{attribute 'GeneratedUsingTerminal: AES-D-BC-ECAT-0000'}
{attribute addProperty BoxType "AES-D-BC-ECAT-0000"}
{attribute addProperty Id "digital_Data_OAT %Q*ARRAY[0..31] OF USINT32"}
{attribute addProperty CRC "2024821696"}
{attribute addProperty Size "32"}
TYPE Outputs_FC2FACAD EXTENDS TcoIo.OutputBase_10CEE7DE :
STRUCT
	{attribute addProperty Name "digital_Data_O"}
	digital_Data_O AT %Q* : ARRAY[0..31] OF USINT;
END_STRUCT
END_TYPE

(* stored: Version 1.2.0.0, ProductVersion 3.1.4024.11
   DUT Outputs_FC2FACAD: Id {39d4f074-f066-0955-3486-5d2418b00f96} *)
